(*			
	RafalOS
	Rafał Osajda		20.11.2025		TC 4024.66
	Interfejs przekazywany do modułów tworzących strony
*)
INTERFACE ITF_MCHMIMachineControl_HMI_PrepScr_07_XX

(*			
	RafalOS
	Rafał Osajda		25.10.2025		TC 4024.66
	Utworzenie nowych szablonów receptur na podstawie dodanych fb zewnętrznych - wywołanie metody powoduje
	skosowanie dotychczasowych szablonów i receptur
*)
METHOD PUBLIC CreateRecipeTemplates : BOOL
VAR_INPUT
END_VAR
END_METHOD

END_INTERFACE

(* stored: Version 1.1.0.1
   Itf ITF_MCHMIMachineControl_HMI_PrepScr_07_XX: Id {b1d637c4-2224-0f0c-3cbe-5dfe517618f2}
   Method CreateRecipeTemplates: Id {312e02d3-defc-0755-3aa3-1ada50e8ad65} *)
